// TIA Portal V19 export
FUNCTION "A01_ButtonsSafe_CALL" : Void   // FC140, LAD
TITLE = BUTTONS SAFE OF AREA 01 CALL
// stored: SetENOAutomatically false
BEGIN

REGION Network 1: LB101
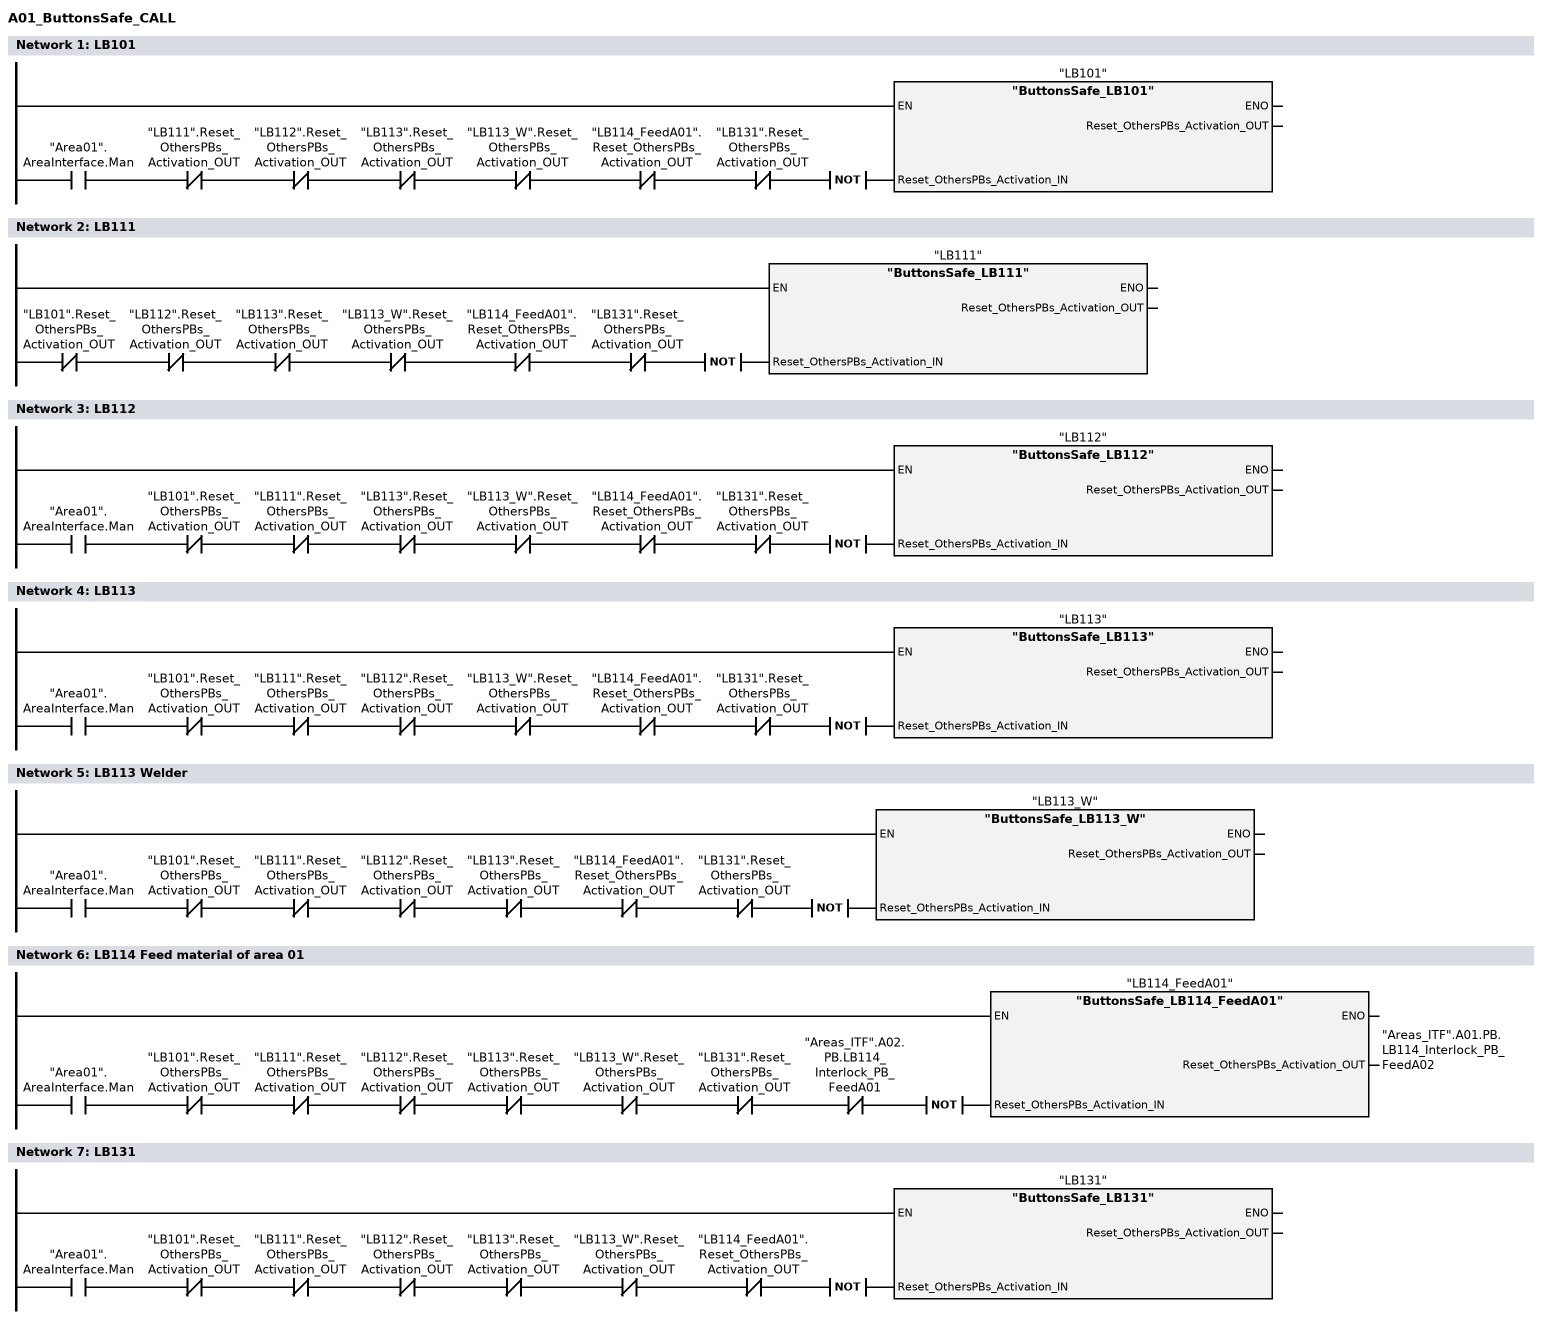
   RUNG wire#powerrail
      "LB101"(Reset_OthersPBs_Activation_IN := wire#w1, Reset_OthersPBs_Activation_OUT =>)
   END_RUNG
   RUNG wire#powerrail
      Contact( "Area01".AreaInterface.Man )
      I_Contact( "LB111".Reset_OthersPBs_Activation_OUT )
      I_Contact( "LB112".Reset_OthersPBs_Activation_OUT )
      I_Contact( "LB113".Reset_OthersPBs_Activation_OUT )
      I_Contact( "LB113_W".Reset_OthersPBs_Activation_OUT )
      I_Contact( "LB114_FeedA01".Reset_OthersPBs_Activation_OUT )
      I_Contact( "LB131".Reset_OthersPBs_Activation_OUT )
      Not()
   END_RUNG wire#w1
   // the same network as SCL:
   "LB101"(Reset_OthersPBs_Activation_IN := NOT ("Area01".AreaInterface.Man AND NOT "LB111".Reset_OthersPBs_Activation_OUT AND NOT "LB112".Reset_OthersPBs_Activation_OUT AND NOT "LB113".Reset_OthersPBs_Activation_OUT AND NOT "LB113_W".Reset_OthersPBs_Activation_OUT AND NOT "LB114_FeedA01".Reset_OthersPBs_Activation_OUT AND NOT "LB131".Reset_OthersPBs_Activation_OUT));   // "ButtonsSafe_LB101"
END_REGION

REGION Network 2: LB111
   RUNG wire#powerrail
      "LB111"(Reset_OthersPBs_Activation_IN := wire#w1, Reset_OthersPBs_Activation_OUT =>)
   END_RUNG
   RUNG wire#powerrail
      I_Contact( "LB101".Reset_OthersPBs_Activation_OUT )
      I_Contact( "LB112".Reset_OthersPBs_Activation_OUT )
      I_Contact( "LB113".Reset_OthersPBs_Activation_OUT )
      I_Contact( "LB113_W".Reset_OthersPBs_Activation_OUT )
      I_Contact( "LB114_FeedA01".Reset_OthersPBs_Activation_OUT )
      I_Contact( "LB131".Reset_OthersPBs_Activation_OUT )
      Not()
   END_RUNG wire#w1
   // the same network as SCL:
   "LB111"(Reset_OthersPBs_Activation_IN := NOT (NOT "LB101".Reset_OthersPBs_Activation_OUT AND NOT "LB112".Reset_OthersPBs_Activation_OUT AND NOT "LB113".Reset_OthersPBs_Activation_OUT AND NOT "LB113_W".Reset_OthersPBs_Activation_OUT AND NOT "LB114_FeedA01".Reset_OthersPBs_Activation_OUT AND NOT "LB131".Reset_OthersPBs_Activation_OUT));   // "ButtonsSafe_LB111"
END_REGION

REGION Network 3: LB112
   RUNG wire#powerrail
      "LB112"(Reset_OthersPBs_Activation_IN := wire#w1, Reset_OthersPBs_Activation_OUT =>)
   END_RUNG
   RUNG wire#powerrail
      Contact( "Area01".AreaInterface.Man )
      I_Contact( "LB101".Reset_OthersPBs_Activation_OUT )
      I_Contact( "LB111".Reset_OthersPBs_Activation_OUT )
      I_Contact( "LB113".Reset_OthersPBs_Activation_OUT )
      I_Contact( "LB113_W".Reset_OthersPBs_Activation_OUT )
      I_Contact( "LB114_FeedA01".Reset_OthersPBs_Activation_OUT )
      I_Contact( "LB131".Reset_OthersPBs_Activation_OUT )
      Not()
   END_RUNG wire#w1
   // the same network as SCL:
   "LB112"(Reset_OthersPBs_Activation_IN := NOT ("Area01".AreaInterface.Man AND NOT "LB101".Reset_OthersPBs_Activation_OUT AND NOT "LB111".Reset_OthersPBs_Activation_OUT AND NOT "LB113".Reset_OthersPBs_Activation_OUT AND NOT "LB113_W".Reset_OthersPBs_Activation_OUT AND NOT "LB114_FeedA01".Reset_OthersPBs_Activation_OUT AND NOT "LB131".Reset_OthersPBs_Activation_OUT));   // "ButtonsSafe_LB112"
END_REGION

REGION Network 4: LB113
   RUNG wire#powerrail
      "LB113"(Reset_OthersPBs_Activation_IN := wire#w1, Reset_OthersPBs_Activation_OUT =>)
   END_RUNG
   RUNG wire#powerrail
      Contact( "Area01".AreaInterface.Man )
      I_Contact( "LB101".Reset_OthersPBs_Activation_OUT )
      I_Contact( "LB111".Reset_OthersPBs_Activation_OUT )
      I_Contact( "LB112".Reset_OthersPBs_Activation_OUT )
      I_Contact( "LB113_W".Reset_OthersPBs_Activation_OUT )
      I_Contact( "LB114_FeedA01".Reset_OthersPBs_Activation_OUT )
      I_Contact( "LB131".Reset_OthersPBs_Activation_OUT )
      Not()
   END_RUNG wire#w1
   // the same network as SCL:
   "LB113"(Reset_OthersPBs_Activation_IN := NOT ("Area01".AreaInterface.Man AND NOT "LB101".Reset_OthersPBs_Activation_OUT AND NOT "LB111".Reset_OthersPBs_Activation_OUT AND NOT "LB112".Reset_OthersPBs_Activation_OUT AND NOT "LB113_W".Reset_OthersPBs_Activation_OUT AND NOT "LB114_FeedA01".Reset_OthersPBs_Activation_OUT AND NOT "LB131".Reset_OthersPBs_Activation_OUT));   // "ButtonsSafe_LB113"
END_REGION

REGION Network 5: LB113 Welder
   RUNG wire#powerrail
      "LB113_W"(Reset_OthersPBs_Activation_IN := wire#w1, Reset_OthersPBs_Activation_OUT =>)
   END_RUNG
   RUNG wire#powerrail
      Contact( "Area01".AreaInterface.Man )
      I_Contact( "LB101".Reset_OthersPBs_Activation_OUT )
      I_Contact( "LB111".Reset_OthersPBs_Activation_OUT )
      I_Contact( "LB112".Reset_OthersPBs_Activation_OUT )
      I_Contact( "LB113".Reset_OthersPBs_Activation_OUT )
      I_Contact( "LB114_FeedA01".Reset_OthersPBs_Activation_OUT )
      I_Contact( "LB131".Reset_OthersPBs_Activation_OUT )
      Not()
   END_RUNG wire#w1
   // the same network as SCL:
   "LB113_W"(Reset_OthersPBs_Activation_IN := NOT ("Area01".AreaInterface.Man AND NOT "LB101".Reset_OthersPBs_Activation_OUT AND NOT "LB111".Reset_OthersPBs_Activation_OUT AND NOT "LB112".Reset_OthersPBs_Activation_OUT AND NOT "LB113".Reset_OthersPBs_Activation_OUT AND NOT "LB114_FeedA01".Reset_OthersPBs_Activation_OUT AND NOT "LB131".Reset_OthersPBs_Activation_OUT));   // "ButtonsSafe_LB113_W"
END_REGION

REGION Network 6: LB114 Feed material of area 01
   RUNG wire#powerrail
      "LB114_FeedA01"(Reset_OthersPBs_Activation_IN := wire#w1, Reset_OthersPBs_Activation_OUT => "Areas_ITF".A01.PB.LB114_Interlock_PB_FeedA02)
   END_RUNG
   RUNG wire#powerrail
      Contact( "Area01".AreaInterface.Man )
      I_Contact( "LB101".Reset_OthersPBs_Activation_OUT )
      I_Contact( "LB111".Reset_OthersPBs_Activation_OUT )
      I_Contact( "LB112".Reset_OthersPBs_Activation_OUT )
      I_Contact( "LB113".Reset_OthersPBs_Activation_OUT )
      I_Contact( "LB113_W".Reset_OthersPBs_Activation_OUT )
      I_Contact( "LB131".Reset_OthersPBs_Activation_OUT )
      I_Contact( "Areas_ITF".A02.PB.LB114_Interlock_PB_FeedA01 )
      Not()
   END_RUNG wire#w1
   // the same network as SCL:
   "LB114_FeedA01"(Reset_OthersPBs_Activation_IN := NOT ("Area01".AreaInterface.Man AND NOT "LB101".Reset_OthersPBs_Activation_OUT AND NOT "LB111".Reset_OthersPBs_Activation_OUT AND NOT "LB112".Reset_OthersPBs_Activation_OUT AND NOT "LB113".Reset_OthersPBs_Activation_OUT AND NOT "LB113_W".Reset_OthersPBs_Activation_OUT AND NOT "LB131".Reset_OthersPBs_Activation_OUT AND NOT "Areas_ITF".A02.PB.LB114_Interlock_PB_FeedA01),   // "ButtonsSafe_LB114_FeedA01"
                   Reset_OthersPBs_Activation_OUT => "Areas_ITF".A01.PB.LB114_Interlock_PB_FeedA02);
END_REGION

REGION Network 7: LB131
   RUNG wire#powerrail
      "LB131"(Reset_OthersPBs_Activation_IN := wire#w1, Reset_OthersPBs_Activation_OUT =>)
   END_RUNG
   RUNG wire#powerrail
      Contact( "Area01".AreaInterface.Man )
      I_Contact( "LB101".Reset_OthersPBs_Activation_OUT )
      I_Contact( "LB111".Reset_OthersPBs_Activation_OUT )
      I_Contact( "LB112".Reset_OthersPBs_Activation_OUT )
      I_Contact( "LB113".Reset_OthersPBs_Activation_OUT )
      I_Contact( "LB113_W".Reset_OthersPBs_Activation_OUT )
      I_Contact( "LB114_FeedA01".Reset_OthersPBs_Activation_OUT )
      Not()
   END_RUNG wire#w1
   // the same network as SCL:
   "LB131"(Reset_OthersPBs_Activation_IN := NOT ("Area01".AreaInterface.Man AND NOT "LB101".Reset_OthersPBs_Activation_OUT AND NOT "LB111".Reset_OthersPBs_Activation_OUT AND NOT "LB112".Reset_OthersPBs_Activation_OUT AND NOT "LB113".Reset_OthersPBs_Activation_OUT AND NOT "LB113_W".Reset_OthersPBs_Activation_OUT AND NOT "LB114_FeedA01".Reset_OthersPBs_Activation_OUT));   // "ButtonsSafe_LB131"
END_REGION

REGION Network 8: >
END_REGION

REGION Network 9: >
END_REGION

REGION Network 10: >
END_REGION
END_FUNCTION
